% RSLogix 500 project I2P Job 15 - Andrew_Hoemmen.RSS, saved by version 10.00.00.00 %
PROJECT "ML03A"    % processor: Bul.1763 MicroLogix 1100 Series B %

PROGRAM FILES
  LAD 2   16 rungs

DATA FILES
  O0 OUTPUT  4 elements
  I1 INPUT  6 elements
  S2 STATUS  66 elements
  B3 BINARY  1 elements
  T4 TIMER  1 elements
  C5 COUNTER  1 elements
  R6 CONTROL  1 elements
  N7 INTEGER  1 elements
  F8 FLOAT  1 elements

LADDER 2
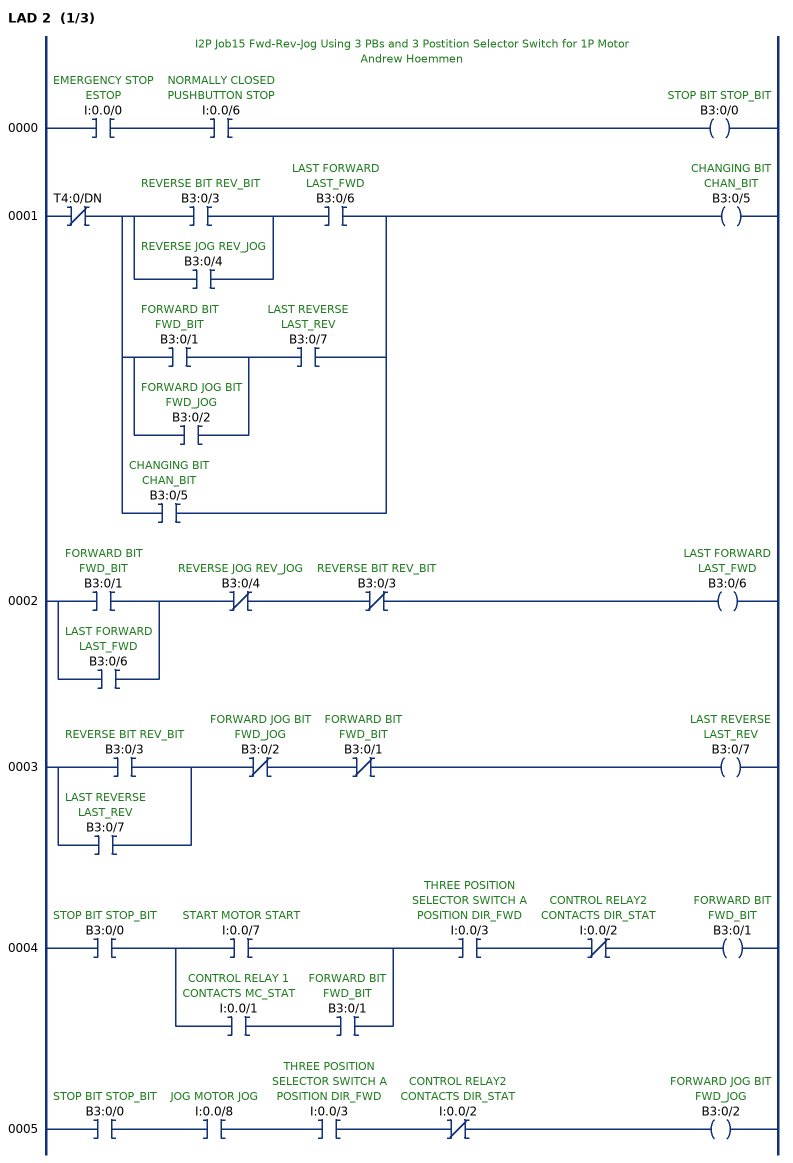
% Rung: 0 %
% I2P Job15 Fwd-Rev-Jog Using 3 PBs and 3 Postition Selector Switch for 1P Motor
% Andrew Hoemmen %
SOR XIC I:0.0/0 XIC I:0.0/6 OTE B3:0/0 EOR
%   I:0.0/0  ESTOP  "EMERGENCY STOP" %
%   I:0.0/6  STOP  "NORMALLY CLOSED PUSHBUTTON" %
%   B3:0/0  STOP_BIT  "STOP BIT" %
% Rung: 1 %
SOR XIO T4:0/DN BST BST XIC B3:0/3 NXB XIC B3:0/4 BND XIC B3:0/6 NXB BST BST XIC B3:0/1 NXB XIC B3:0/2 BND XIC B3:0/7 NXB XIC B3:0/5 BND BND OTE B3:0/5 EOR
%   B3:0/3  REV_BIT  "REVERSE BIT" %
%   B3:0/4  REV_JOG  "REVERSE JOG" %
%   B3:0/6  LAST_FWD  "LAST FORWARD" %
%   B3:0/1  FWD_BIT  "FORWARD BIT" %
%   B3:0/2  FWD_JOG  "FORWARD JOG BIT" %
%   B3:0/7  LAST_REV  "LAST REVERSE" %
%   B3:0/5  CHAN_BIT  "CHANGING BIT" %
% Rung: 2 %
SOR BST XIC B3:0/1 NXB XIC B3:0/6 BND XIO B3:0/4 XIO B3:0/3 OTE B3:0/6 EOR
%   B3:0/1  FWD_BIT  "FORWARD BIT" %
%   B3:0/6  LAST_FWD  "LAST FORWARD" %
%   B3:0/4  REV_JOG  "REVERSE JOG" %
%   B3:0/3  REV_BIT  "REVERSE BIT" %
% Rung: 3 %
SOR BST XIC B3:0/3 NXB XIC B3:0/7 BND XIO B3:0/2 XIO B3:0/1 OTE B3:0/7 EOR
%   B3:0/3  REV_BIT  "REVERSE BIT" %
%   B3:0/7  LAST_REV  "LAST REVERSE" %
%   B3:0/2  FWD_JOG  "FORWARD JOG BIT" %
%   B3:0/1  FWD_BIT  "FORWARD BIT" %
% Rung: 4 %
SOR XIC B3:0/0 BST XIC I:0.0/7 NXB XIC I:0.0/1 XIC B3:0/1 BND XIC I:0.0/3 XIO I:0.0/2 OTE B3:0/1 EOR
%   B3:0/0  STOP_BIT  "STOP BIT" %
%   I:0.0/7  START  "START MOTOR" %
%   I:0.0/1  MC_STAT  "CONTROL RELAY 1 CONTACTS" %
%   B3:0/1  FWD_BIT  "FORWARD BIT" %
%   I:0.0/3  DIR_FWD  "THREE POSITION SELECTOR SWITCH A POSITION" %
%   I:0.0/2  DIR_STAT  "CONTROL RELAY2 CONTACTS" %
% Rung: 5 %
SOR XIC B3:0/0 XIC I:0.0/8 XIC I:0.0/3 XIO I:0.0/2 OTE B3:0/2 EOR
%   B3:0/0  STOP_BIT  "STOP BIT" %
%   I:0.0/8  JOG  "JOG MOTOR" %
%   I:0.0/3  DIR_FWD  "THREE POSITION SELECTOR SWITCH A POSITION" %
%   I:0.0/2  DIR_STAT  "CONTROL RELAY2 CONTACTS" %
%   B3:0/2  FWD_JOG  "FORWARD JOG BIT" %

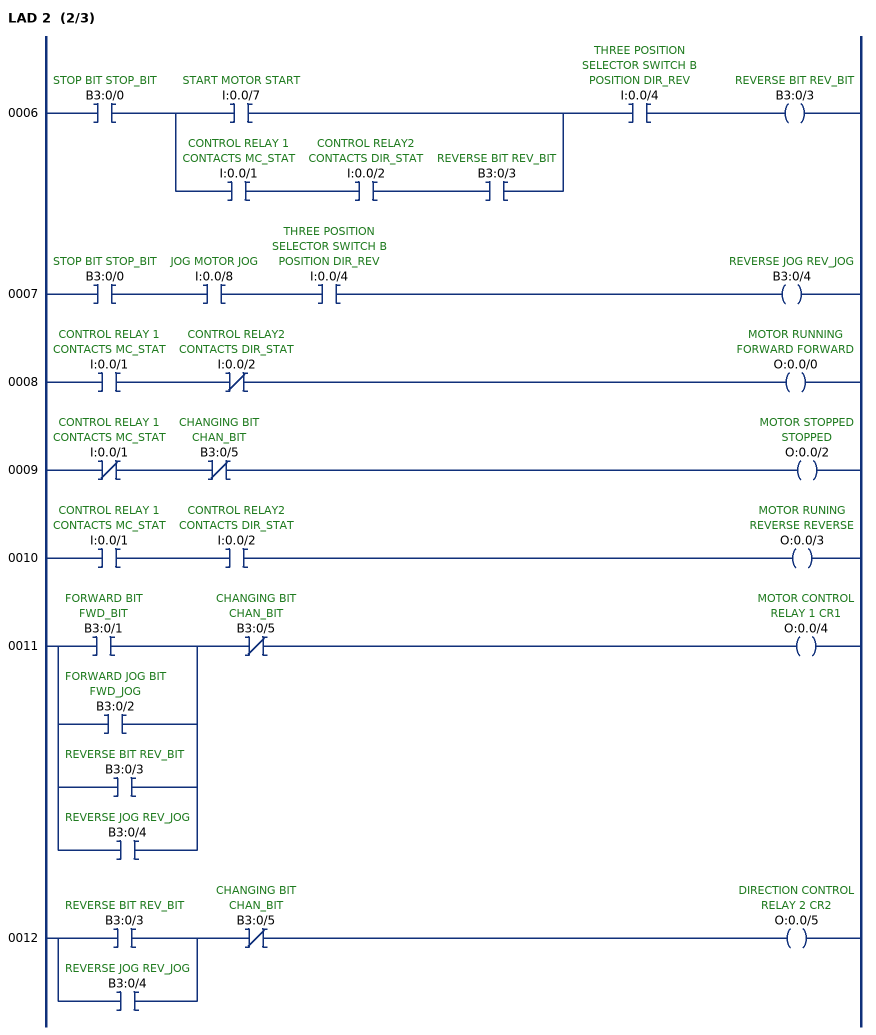
% Rung: 6 %
SOR XIC B3:0/0 BST XIC I:0.0/7 NXB XIC I:0.0/1 XIC I:0.0/2 XIC B3:0/3 BND XIC I:0.0/4 OTE B3:0/3 EOR
%   B3:0/0  STOP_BIT  "STOP BIT" %
%   I:0.0/7  START  "START MOTOR" %
%   I:0.0/1  MC_STAT  "CONTROL RELAY 1 CONTACTS" %
%   I:0.0/2  DIR_STAT  "CONTROL RELAY2 CONTACTS" %
%   B3:0/3  REV_BIT  "REVERSE BIT" %
%   I:0.0/4  DIR_REV  "THREE POSITION SELECTOR SWITCH B POSITION" %
% Rung: 7 %
SOR XIC B3:0/0 XIC I:0.0/8 XIC I:0.0/4 OTE B3:0/4 EOR
%   B3:0/0  STOP_BIT  "STOP BIT" %
%   I:0.0/8  JOG  "JOG MOTOR" %
%   I:0.0/4  DIR_REV  "THREE POSITION SELECTOR SWITCH B POSITION" %
%   B3:0/4  REV_JOG  "REVERSE JOG" %
% Rung: 8 %
SOR XIC I:0.0/1 XIO I:0.0/2 OTE O:0.0/0 EOR
%   I:0.0/1  MC_STAT  "CONTROL RELAY 1 CONTACTS" %
%   I:0.0/2  DIR_STAT  "CONTROL RELAY2 CONTACTS" %
%   O:0.0/0  FORWARD  "MOTOR RUNNING FORWARD" %
% Rung: 9 %
SOR XIO I:0.0/1 XIO B3:0/5 OTE O:0.0/2 EOR
%   I:0.0/1  MC_STAT  "CONTROL RELAY 1 CONTACTS" %
%   B3:0/5  CHAN_BIT  "CHANGING BIT" %
%   O:0.0/2  STOPPED  "MOTOR STOPPED" %
% Rung: 10 %
SOR XIC I:0.0/1 XIC I:0.0/2 OTE O:0.0/3 EOR
%   I:0.0/1  MC_STAT  "CONTROL RELAY 1 CONTACTS" %
%   I:0.0/2  DIR_STAT  "CONTROL RELAY2 CONTACTS" %
%   O:0.0/3  REVERSE  "MOTOR RUNING REVERSE" %
% Rung: 11 %
SOR BST XIC B3:0/1 NXB BST XIC B3:0/2 NXB BST XIC B3:0/3 NXB XIC B3:0/4 BND BND BND XIO B3:0/5 OTE O:0.0/4 EOR
%   B3:0/1  FWD_BIT  "FORWARD BIT" %
%   B3:0/2  FWD_JOG  "FORWARD JOG BIT" %
%   B3:0/3  REV_BIT  "REVERSE BIT" %
%   B3:0/4  REV_JOG  "REVERSE JOG" %
%   B3:0/5  CHAN_BIT  "CHANGING BIT" %
%   O:0.0/4  CR1  "MOTOR CONTROL RELAY 1" %
% Rung: 12 %
SOR BST XIC B3:0/3 NXB XIC B3:0/4 BND XIO B3:0/5 OTE O:0.0/5 EOR
%   B3:0/3  REV_BIT  "REVERSE BIT" %
%   B3:0/4  REV_JOG  "REVERSE JOG" %
%   B3:0/5  CHAN_BIT  "CHANGING BIT" %
%   O:0.0/5  CR2  "DIRECTION CONTROL RELAY 2" %

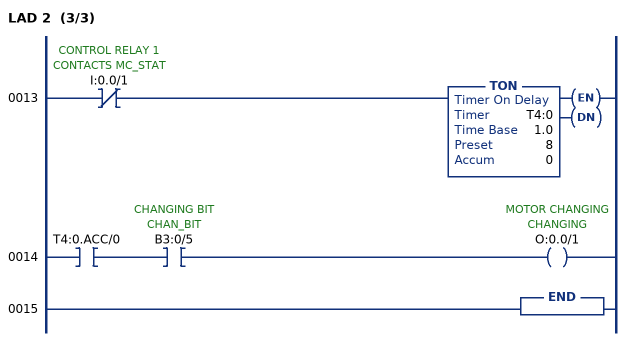
% Rung: 13 %
SOR XIO I:0.0/1 TON T4:0 1.0 8 0 EOR
%   I:0.0/1  MC_STAT  "CONTROL RELAY 1 CONTACTS" %
% Rung: 14 %
SOR XIC T4:0.ACC/0 XIC B3:0/5 OTE O:0.0/1 EOR
%   B3:0/5  CHAN_BIT  "CHANGING BIT" %
%   O:0.0/1  CHANGING  "MOTOR CHANGING" %
% Rung: 15 %
SOR END EOR

OTHER DOCUMENTED ADDRESSES
  DIR_STATS  
  I:0.0/5  2PSS  "TWO POSITION SELECTOR SWITCH"
  T4:0.ACC  BLINK  "LIGHT BLINKING"

DATA TABLE (non-zero values as saved)
DATA T4
% .PRE .ACC %
% T4:0 % 8 0
